FUNCTION IsSome : BOOL
VAR_INPUT
	nIn				: Result;
END_VAR
VAR_OUTPUT
	nOut			: Result;
END_VAR

IsSome := nIn <> 0;
nOut := nIn;

END_FUNCTION

(* stored: Version 1.1.0.1
   POU IsSome: Id {8bd0ebbc-727e-4638-b872-a07d8f4548db}, SpecialFunc None *)
